RoboDK station: limpialados.rdk

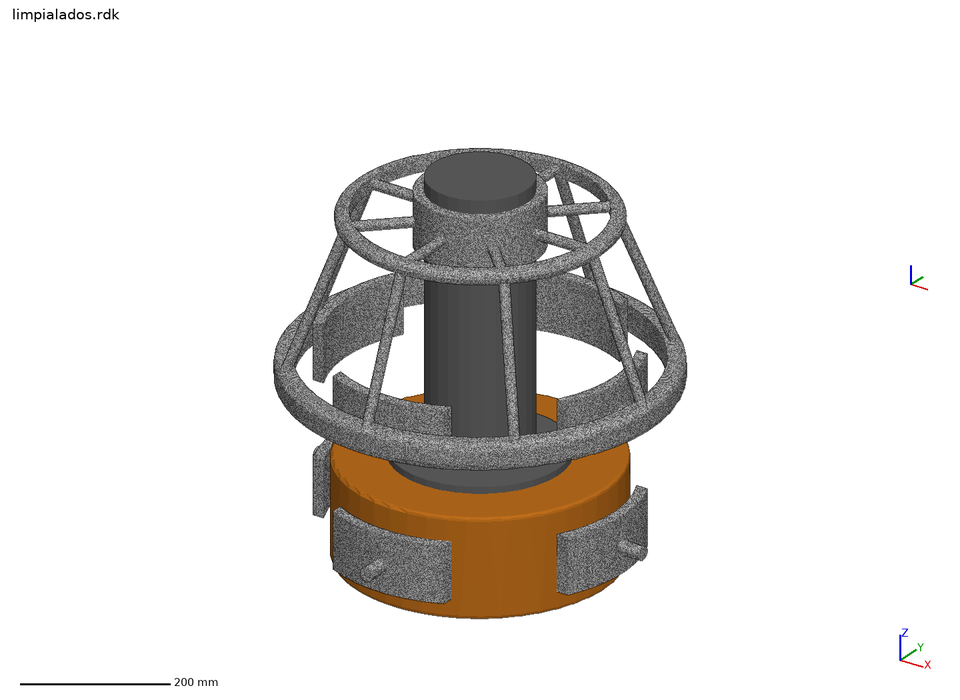
[picture v0: the station drawn from its stored meshes, robots at their saved joint values, targets as dots, program paths as lines]
Station limpialados (saved by RoboDK 5.8.0). Poses are relative to the parent item; angles as X-Y-Z fixed-axis rotations.
  - object eje at (0, 1000, 0) mm, size 250 x 250 x 410 mm, geometry from eje.step
  - object queso at (0, 1000, 0) mm, size 400 x 399.8 x 150 mm, geometry from queso.step
  - object cepillo1 at (0, 0, 0) mm, size 182.2 x 74.5 x 85.5 mm, geometry from cepillo.step
  - object cepillo2 at (0, 0, 0) mm, rotated rx 0 ry 0 rz 90 deg, size 182.2 x 74.5 x 85.5 mm, geometry from cepillo.step
  - object cepillo3 at (0, 0, 0) mm, rotated rx 0 ry 0 rz 180 deg, size 182.2 x 74.5 x 85.5 mm, geometry from cepillo.step
  - object cepillo4 at (0, 0, 0) mm, rotated rx 0 ry 0 rz -90 deg, size 182.2 x 74.5 x 85.5 mm, geometry from cepillo.step
  - frame cep3 at (0, 2000, 0) mm
    - robot cep3: 1 axes
        modified DH rows (alpha deg, a mm, theta deg, d mm): 0, 0, 0, 0 linear
        base shift (0, 0, 0) mm, rotated rx 0 ry 90 rz 90 deg
        joint limits [-15] to [0]; home [0]; saved at [0]
  - object Eje rotatorio cilindro at (0, 1000, 0) mm, size 550 x 549.8 x 285 mm, geometry from Eje rotatorio cilindro  (1).step
  - frame cep2 at (0, 3000, 0) mm
    - robot cep2: 1 axes
        modified DH rows (alpha deg, a mm, theta deg, d mm): 0, 0, 0, 0 linear
        base shift (0, 0, 0) mm, rotated rx 0 ry 90 rz 0 deg
        joint limits [-15] to [0]; home [0]; saved at [0]
  - frame cep4 at (0, 4000, 0) mm
    - robot cep4: 1 axes
        modified DH rows (alpha deg, a mm, theta deg, d mm): 0, 0, 0, 0 linear
        base shift (0, 0, 0) mm, rotated rx 0 ry 90 rz 0 deg
        joint limits [0] to [15]; home [0]; saved at [0]
  - frame cep1 at (0, 5000, 0) mm
    - robot cep1: 1 axes
        modified DH rows (alpha deg, a mm, theta deg, d mm): 0, 0, 0, 0 linear
        base shift (0, 0, 0) mm, rotated rx 0 ry 90 rz 90 deg
        joint limits [0] to [15]; home [0]; saved at [0]
  - object tim at (0, 1000, 200) mm, size 550 x 549.8 x 305 mm, geometry from timón abierto.step
  - object tim at (0, 1000, 0) mm, size 550 x 549.8 x 305 mm, geometry from timón cerrado.step
  - frame timón abierto at (0, 6000, 0) mm
    - robot tim: 1 axes
        modified DH rows (alpha deg, a mm, theta deg, d mm): 0, 0, 0, 0 linear
        joint limits [-35] to [200]; home [0]; saved at [200]
  - Python program Prog1 (listed below)
  - Python program prueba (listed below)
  - object queso2 at (0, 0, 0) mm, size 400 x 399.8 x 150 mm, geometry from queso.step

--- Python program Prog1 ---
import time  # Importar el módulo time para usar sleep
from robodk.robolink import *  # API principal de RoboDK
from robodk.robomath import *  # API principal de RoboDK



# Conectar con RoboDK
RDK = Robolink()

# Obtener los elementos necesarios
timon_a = RDK.Item('timón abierto', ITEM_TYPE_ROBOT)
cep1 = RDK.Item('cep1', ITEM_TYPE_ROBOT)
cep2 = RDK.Item('cep2', ITEM_TYPE_ROBOT)
cep3 = RDK.Item('cep3', ITEM_TYPE_ROBOT)
cep4 = RDK.Item('cep4', ITEM_TYPE_ROBOT)

timon_comp = RDK.Item('Eje rotatorio cilindro', ITEM_TYPE_OBJECT)

# ----------------------
# Verificar el robot 'timón abierto'

art_timon_a = timon_a.Joints()


posicion_actual = art_timon_a[0,0]  # Obtener la primera articulación
nueva_posicion = posicion_actual - 200  # Nueva posición calculada
nueva_posicion = float(nueva_posicion)
# Mover el robot y devolverlo a la posición original
timon_a.MoveJ([nueva_posicion], blocking=True)
#timon_a.MoveJ([posicion_actual], blocking=True)


# ----------------------Cepillos
timon_comp.setVisible(True)
timon_a.setVisible(False)

cep1.setVisible(True)
cep2.setVisible(True)
cep3.setVisible(True)
cep4.setVisible(True)



art_cep1 = cep1.Joints()
art_cep2 = cep2.Joints()
art_cep3 = cep3.Joints()
art_cep4 = cep4.Joints()


posicion_actual_cep1 = art_cep1[0,0]
nueva_posicion_cep1 = posicion_actual_cep1 + 15
nueva_posicion_cep1 = float(nueva_posicion_cep1)

posicion_actual_cep2 = art_cep2[0,0]
nueva_posicion_cep2 = posicion_actual_cep2 - 15
nueva_posicion_cep2 = float(nueva_posicion_cep2)

posicion_actual_cep3 = art_cep3[0,0]
nueva_posicion_cep3 = posicion_actual_cep3 - 15
nueva_posicion_cep3 = float(nueva_posicion_cep3)

posicion_actual_cep4 = art_cep4[0,0]
nueva_posicion_cep4 = posicion_actual_cep4 + 15
nueva_posicion_cep4 = float(nueva_posicion_cep4)



cep1.setSpeed(10, 0)
cep1.MoveJ([nueva_posicion_cep1], blocking=False)
cep2.setSpeed(10, 0)
cep2.MoveJ([nueva_posicion_cep2], blocking=False)
cep3.setSpeed(10, 0)
cep3.MoveJ([nueva_posicion_cep3], blocking=False)
cep4.setSpeed(10, 0)
cep4.MoveJ([nueva_posicion_cep4], blocking=False)


time.sleep(0.5)
# Seleccionar el objeto a mover
timon_c = RDK.Item('timón cerrado', ITEM_TYPE_OBJECT)
timon_c.setVisible(True)
timon_comp.setVisible(False)
cep1.setVisible(False)
cep2.setVisible(False)
cep3.setVisible(False)
cep4.setVisible(False)

time.sleep(0.5)



    # Obtener la pose actual del objeto

incremento = 1
# Movimiento
# Traslación de 0.001 mm cada milisegundo en el eje Z
desplazamiento = transl(0, 0, incremento)

# Rotación de 1 grado cada milisegundo alrededor del eje Z
rotacion = rotz(0.1)  # 0.1 grados por milisegundo (puedes ajustar)

for t in range(360):  # 5 segundos a 1000 milisegundos
    pose_actual = timon_c.Pose()

    if t < 30:
        incremento = 1
    elif t < 90:
        incremento = -1
    elif t < 150:
        incremento = 1
    elif t < 210:
        incremento = -1
    elif t < 270:
        incremento = 1
    elif t < 330:
        incremento = -1
    else:
        incremento = 1

    desplazamiento = transl(0, 0, incremento)


    nueva_pose = pose_actual * desplazamiento * rotacion


    # Establecer la nueva pose del objeto
    timon_c.setPose(nueva_pose)

    # Esperar 1 milisegundo
    time.sleep(0.001)

pose_a_copiar = timon_comp.Pose()
timon_c.setPose(pose_a_copiar)
time.sleep(0.5)
timon_comp.setVisible(True)
cep1.setVisible(True)
cep2.setVisible(True)
cep3.setVisible(True)
cep4.setVisible(True)
timon_c.setVisible(False)

cep1.MoveJ([posicion_actual_cep1], blocking=False)
cep2.MoveJ([posicion_actual_cep2], blocking=False)
cep3.MoveJ([posicion_actual_cep3], blocking=False)
cep4.MoveJ([posicion_actual_cep4], blocking=False)

time.sleep(0.2)

timon_a.setVisible(True)
time.sleep(0.1)
timon_comp.setVisible(False)
cep1.setVisible(False)
cep2.setVisible(False)
cep3.setVisible(False)
cep4.setVisible(False)

timon_a.MoveJ([posicion_actual], blocking=True)

--- Python program prueba ---
import time
from robodk.robolink import *  # API principal de RoboDK
from robodk.robomath import *  # API de matemáticas (transformaciones)

# Conectar con RoboDK
RDK = Robolink()

# Seleccionar el objeto a mover
timon_c = RDK.Item('timón cerrado', ITEM_TYPE_OBJECT)

# Comprobar si el objeto es válido
if not timon_c.Valid():
    print("Error: El objeto no fue encontrado en el proyecto.")
else:
    # Obtener la pose actual del objeto

    incremento = 1
    # Movimiento
    # Traslación de 0.001 mm cada milisegundo en el eje Z
    desplazamiento = transl(0, 0, incremento)

    # Rotación de 1 grado cada milisegundo alrededor del eje Z
    rotacion = rotz(0.1)  # 0.1 grados por milisegundo (puedes ajustar)

    for t in range(300):  # 5 segundos a 1000 milisegundos
        pose_actual = timon_c.Pose()

        if t < 30:
            incremento = 1
        elif t < 90:
            incremento = -1
        elif t < 150:
            incremento = 1
        elif t < 210:
            incremento = -1
        elif t < 270:
            incremento = 1
        else:
            incremento = -1


        desplazamiento = transl(0, 0, incremento)

        nueva_pose = pose_actual * desplazamiento * rotacion

        # Establecer la nueva pose del objeto
        timon_c.setPose(nueva_pose)

        # Esperar 1 milisegundo
        time.sleep(0.001)

    print("El objeto ha terminado de moverse y rotar.")
